// TIA Portal V19 export
DATA_BLOCK "A0303_Sostegno_Coda"   // DB94
// stored: InstanceOfName A0303_Sostegno_FB, InstanceOfType FB
"A0303_Sostegno_FB"
   // VAR_INPUT
   //    AreaInterface : "AreaInterface";
   //    ZSI : "udt_ZoneSafetyInterface";
   //    DSI_Feed : "udt_DeviceSafetyInterface";
   //    DSI_Valve : "udt_DeviceSafetyInterface";
   //    DataIn : Struct
   //       OP_Work_PB : Bool;
   //       OP_Rest_PB : Bool;
   //       Pos0_Ls : Bool;
   //       Pos1_Ls : Bool;
   //       Pos2_Ls : Bool;
   //    END_STRUCT;
   //    CIn : Struct
   //       Manager : Struct
   //          EnableStopDoorOpeningReq : Bool;
   //          EnableStopInPhase : Bool;
   //          EnableStopProgrammed : Bool;
   //          Control_ON : Bool;
   //          CanMoveFreely : Bool;
   //          Phase : Struct
   //             VAI_A_LAVORO : Bool;
   //             VAI_A_RIPOSO : Bool;
   //          END_STRUCT;
   //          Ax : Struct
   //             Pos { ExternalVisible := 'False'; ExternalWritable := 'False'} : LReal;
   //          END_STRUCT;
   //          Paletti : Struct
   //             PosPaletto : Int;
   //             Pos1Collision : Bool;
   //             Pos2Collision : Bool;
   //          END_STRUCT;
   //       END_STRUCT;
   //       Navetta : Struct
   //          OutOfWorkspace : Bool;
   //       END_STRUCT;
   //       Trasporto : Struct
   //          OutOfWorkspace : Bool;
   //       END_STRUCT;
   //       CycleModeShortPiece : Bool;
   //    END_STRUCT;
   //    Config : Struct
   //       Ax : "Positioning_DOL_Machine_Config";
   //       V_1 : "ValveMachine_Config";
   //       V_2 : "ValveMachine_Config";
   //       DelayMissingCondition { ExternalAccessible := 'False'; ExternalVisible := 'False'; ExternalWritable := 'False'} : Time;
   //    END_STRUCT;
   //    HWID : Struct
   //       Ax_TEL1 : HW_SUBMODULE;
   //       Enc_IO : HW_SUBMODULE;
   //    END_STRUCT;
   // END_VAR
   // VAR_OUTPUT
   //    MachineInterface : "MachineInterface";
   //    COut : Struct
   //       Ax : "Positioning_DOL_Machine_COut";
   //       Paletto : Struct
   //          CtrlSafe : Bool;
   //          Standstill : Bool;
   //          Rest_CheckNext : Bool;
   //          Work_CheckNext : Bool;
   //          Pos : Int;
   //          RestPosition : Bool;
   //       END_STRUCT;
   //    END_STRUCT;
   // END_VAR
   // VAR_IN_OUT
   //    Par : Struct
   //       Ax : "Positioning_DOL_Machine_Par";
   //       Ax_Pers : "Positioning_DOL_Machine_Pers_Data";
   //       Enc : "PosFbk_RTN";
   //    END_STRUCT;
   //    Par_Mach : Struct
   //       RestPosition : LReal;
   //       ToleranceWindow : LReal;
   //       PosTimeout : Time;
   //    END_STRUCT;
   // END_VAR
   // VAR
   //    Alarm : Struct
   //       Ax { S7_SetPoint := 'True'} : "Positioning_DOL_Machine_Alr";
   //       V_1 : "ValveAlr";
   //       V_2 : "ValveAlr";
   //       Enc { S7_SetPoint := 'True'} : "PosFbk_Encoder_Alr";
   //       Missing_Pos0_Ls_ON { S7_SetPoint := 'True'} : Bool;
   //       Missing_Pos1_Ls_ON { S7_SetPoint := 'True'} : Bool;
   //       Missing_Pos2_Ls_ON { S7_SetPoint := 'True'} : Bool;
   //       LimitSwitch : Bool;
   //    END_STRUCT;
   //    Warning : Struct
   //       Ax { S7_SetPoint := 'True'} : "Positioning_DOL_Machine_Wng";
   //       V_1 { S7_SetPoint := 'True'} : "ValveMachine_Wng";
   //       V_2 { S7_SetPoint := 'True'} : "ValveMachine_Wng";
   //       V_Paletti { S7_SetPoint := 'True'} : "ValveMachine_Wng";
   //       MissingCnd : Struct
   //          OP_REST : Bool;
   //          OP_WORK : Bool;
   //          AxInRestPos : Bool;
   //       END_STRUCT;
   //    END_STRUCT;
   //    Ctrl : Struct
   //       Man : Struct
   //          OP_Vai_A_Lavoro : Bool;
   //          OP_Vai_A_Riposo : Bool;
   //       END_STRUCT;
   //       Aut : Struct
   //          OP_Vai_A_Lavoro : Bool;
   //          OP_Vai_A_Riposo : Bool;
   //       END_STRUCT;
   //       Pos0 : Bool;
   //       Pos1 : Bool;
   //       Pos2 : Bool;
   //       OP_Vai_A_Lavoro : Bool;
   //       OP_Vai_A_Riposo : Bool;
   //    END_STRUCT;
   //    Sts : Struct
   //       OP_Ax_CanMoveFreely : Bool;
   //       OP_CanMoveFreely : Bool;
   //       OP_Rest_Cnd : Bool;
   //       OP_Work_Cnd : Bool;
   //       InRestPos : Bool;
   //    END_STRUCT;
   //    HMI : Struct
   //       PbPreset : Bool;
   //       PresetValue : LReal;
   //    END_STRUCT;
   //    Ax { S7_SetPoint := 'True'} : "Positioning_DOL_Machine_FB";
   //    Enc : "PosFbk_SickAFM60";
   //    Enc_ITF : "PosFbk_ITF";
   //    V_1 { S7_SetPoint := 'True'} : "ValveMachine_FB";
   //    V_2 { S7_SetPoint := 'True'} : "ValveMachine_FB";
   //    AUX : Struct
   //       OP_Work_PB { ExternalAccessible := 'False'; ExternalVisible := 'False'; ExternalWritable := 'False'} : Bool;
   //       OP_Rest_PB { ExternalAccessible := 'False'; ExternalVisible := 'False'; ExternalWritable := 'False'} : Bool;
   //       OP_MoveToPos : Bool;
   //       PbPos0 : Bool;
   //       PbPos1 : Bool;
   //       PbPos2 : Bool;
   //    END_STRUCT;
   //    TON_MissingLsPos0 : IEC_TIMER;
   //    TON_MissingLsPos1 : IEC_TIMER;
   //    TON_MissingLsPos2 : IEC_TIMER;
   //    TON_OP_REST_MissingCnd : IEC_TIMER;
   //    TON_OP_WORK_MissingCnd : IEC_TIMER;
   // END_VAR
BEGIN
END_DATA_BLOCK
